{attribute addProperty BoxType "EJ2521-0224-0016"}
{attribute addProperty Id "Enable_latch_extern_on_positive_edgeBIT10.1252Set_counterBIT10.1253Enable_latch_extern_on_negative_edgeBIT10.1254"}
{attribute addProperty CRC "3903845343"}
{attribute addProperty SizeInBites "16"}
{attribute addProperty SizeInBytes "2"}
TYPE Control_E8AFF3DF :
STRUCT
	{attribute 'hide'}
	reserve_1 : BIT;
	{attribute addProperty Name "Enable_latch_extern_on_positive_edge"}
	Enable_latch_extern_on_positive_edge : BIT;
	{attribute addProperty Name "Set_counter"}
	Set_counter : BIT;
	{attribute addProperty Name "Enable_latch_extern_on_negative_edge"}
	Enable_latch_extern_on_negative_edge : BIT;
	{attribute 'hide'}
	reserve_2_BIT_0 : BIT;
	{attribute 'hide'}
	reserve_2_BIT_1 : BIT;
	{attribute 'hide'}
	reserve_2_BIT_2 : BIT;
	{attribute 'hide'}
	reserve_2_BIT_3 : BIT;
	{attribute 'hide'}
	reserve_3 : BYTE;
END_STRUCT
END_TYPE

(* stored: Version 1.2.0.0, ProductVersion 3.1.4024.9
   DUT Control_E8AFF3DF: Id {e895ce8b-562c-4024-a1d4-8235c813c4a5} *)
